// TwinCAT 3 PLC project Dbg
// Title: Debug
// Company: _
// Author: Krystian Lis et al.
// ProjectVersion: 1.0.0
// Description: Code debugging helper.
// ProgramVersion: 3.1.4026.9
// libraries:
//   Strings, * (_)
// project tree:
//   Dbg/ DebugMsg.TcPOU, DebugList.TcPOU, DebugLen.TcPOU, I_Debug.TcIO, Param.TcGVL, ST_DebugInfo.TcDUT, _Debug.TcGVL

// ---- Dbg/ST_DebugInfo.TcDUT
TYPE INTERNAL ST_DebugInfo :
STRUCT
	iDebug		: I_Debug;
	sInfo		: Strings.Str;
END_STRUCT
END_TYPE

// ---- Dbg/Param.TcGVL
{attribute 'qualified_only'}
VAR_GLOBAL CONSTANT
	nMaxDebugArraySize		: UDINT := 10;
END_VAR

// ---- Dbg/_Debug.TcGVL
{attribute 'qualified_only'}
VAR_GLOBAL INTERNAL
	stDebug				: ARRAY[0..Param.nMaxDebugArraySize] OF ST_DebugInfo;
	nDebugLen			: UDINT;	
END_VAR

// ---- Dbg/I_Debug.TcIO
INTERFACE I_Debug

END_INTERFACE

// ---- Dbg/DebugMsg.TcPOU
FUNCTION DebugMsg
VAR_INPUT
	iDebug			: I_Debug;
	sInfo			: Strings.Str;
END_VAR
VAR
END_VAR

IF _Debug.nDebugLen = Param.nMaxDebugArraySize THEN
	RETURN;	
ELSIF _Debug.nDebugLen = Param.nMaxDebugArraySize - 1 THEN
	_Debug.stDebug[_Debug.nDebugLen].iDebug := 0;
	_Debug.stDebug[_Debug.nDebugLen].sInfo := 'Debug overflow!';
	RETURN;
END_IF

_Debug.stDebug[_Debug.nDebugLen].iDebug := iDebug;
_Debug.stDebug[_Debug.nDebugLen].sInfo := sInfo;
_Debug.nDebugLen := _Debug.nDebugLen + 1;

END_FUNCTION

// ---- Dbg/DebugList.TcPOU
FUNCTION_BLOCK DebugList
VAR
	_refDebug			: REFERENCE TO ARRAY[0..Param.nMaxDebugArraySize] OF ST_DebugInfo REF= _Debug.stDebug;
END_VAR

END_FUNCTION_BLOCK

// ---- Dbg/DebugLen.TcPOU
FUNCTION DebugLen : UDINT

DebugLen := _Debug.nDebugLen;

END_FUNCTION
